// TIA Portal V16 export
// export: Created 2024-02-03T19:53:39.3632235Z, ExportSetting WithDefaults, DisplayName Totally Integrated Automation Portal, DisplayVersion V16 Update 6, DisplayName TIA Portal Version Control Interface, DisplayVersion V16 Update 2, DisplayName TIA Portal Openness, DisplayVersion V16 Update 6, DisplayName SINAMICS Startdrive Advanced, DisplayVersion V16 Update 5, DisplayName SINAMICS Startdrive G130, G150, S120, S150, SINAMICS MV, S210, DisplayVersion V16 Update 5, DisplayName SINAMICS Startdrive G110M, G120, G120C, G120D, G120P, G115D, DisplayVersion V16 Update 5, DisplayName STEP 7 Professional, DisplayVersion V16 Update 6, DisplayName STEP 7 Safety, DisplayVersion V16, DisplayName WinCC Professional, DisplayVersion V16 Update 6
VAR_GLOBAL   // PLC tag table "Default tag table"
   System_Byte AT %MB1 : Byte;
   FirstScan AT %M1.0 : Bool;
   DiagStatusUpdate AT %M1.1 : Bool;
   AlwaysTRUE AT %M1.2 : Bool;
   AlwaysFALSE AT %M1.3 : Bool;
   Clock_Byte AT %MB0 : Byte;
   Clock_10Hz AT %M0.0 : Bool;
   Clock_5Hz AT %M0.1 : Bool;
   "Clock_2.5Hz" AT %M0.2 : Bool;
   Clock_2Hz AT %M0.3 : Bool;
   "Clock_1.25Hz" AT %M0.4 : Bool;
   Clock_1Hz AT %M0.5 : Bool;
   "Clock_0.625Hz" AT %M0.6 : Bool;
   "Clock_0.5Hz" AT %M0.7 : Bool;
   PositioningAxis_1_Actor_Interface_AddressIn AT %I0.0 : "PD_TEL105_IN";
   PositioningAxis_1_Actor_Interface_AddressOut AT %Q0.0 : "PD_TEL105_OUT";
   PositioningAxis_1_Actor_Interface_TorqueDataAddressIn AT %I40.0 : "PD_TEL750_IN";
   PositioningAxis_1_Actor_Interface_TorqueDataAddressOut AT %Q40.0 : "PD_TEL750_OUT";
   "PositioningAxis_1_Actor_Interface_TorqueDataAddressIn(1)" AT %I44.0 : "PD_TEL750_IN";
   "PositioningAxis_1_Actor_Interface_TorqueDataAddressOut(1)" AT %Q52.0 : "PD_TEL750_OUT";
   SynchronousAxis_1_Actor_Interface_AddressIn AT %I20.0 : "PD_TEL105_IN";
   SynchronousAxis_1_Actor_Interface_AddressOut AT %Q20.0 : "PD_TEL105_OUT";
   SynchronousAxis_1_Actor_Interface_TorqueDataAddressIn AT %I42.0 : "PD_TEL750_IN";
   SynchronousAxis_1_Actor_Interface_TorqueDataAddressOut AT %Q46.0 : "PD_TEL750_OUT";
   "SynchronousAxis_1_Actor_Interface_TorqueDataAddressIn(1)" AT %I46.0 : "PD_TEL750_IN";
   "SynchronousAxis_1_Actor_Interface_TorqueDataAddressOut(1)" AT %Q58.0 : "PD_TEL750_OUT";
END_VAR
